// TIA Portal V16 export
// export: Created 2024-12-03T15:41:44.9252202Z, ExportSetting WithReadOnly, DisplayName Totally Integrated Automation Portal, DisplayVersion V16 Update 6, DisplayName TIA Portal Version Control Interface, DisplayVersion V16 Update 2, DisplayName TIA Portal Openness, DisplayVersion V16 Update 6, DisplayName TIA Portal Teamcenter Gateway, DisplayVersion V16, DisplayName SINAMICS Startdrive Advanced, DisplayVersion V16 Update 5, DisplayName SINAMICS Startdrive G130, G150, S120, S150, SINAMICS MV, S210, DisplayVersion V16 Update 5, DisplayName SINAMICS Startdrive G110M, G120, G120C, G120D, G120P, G115D, DisplayVersion V16 Update 5, DisplayName STEP 7 Professional, DisplayVersion V16 Update 6, DisplayName STEP 7 Safety, DisplayVersion V16, DisplayName WinCC Advanced / Unified PC, DisplayVersion V16 Update 6
TYPE "CLXAiPLC_OUT_UDT"
// stored: CreationDate 2021-07-13T07:41:36.2278727Z, InterfaceModifiedDate 2019-12-05T06:54:01.7617053Z, IsConsistent true, LibraryConformanceStatus The object is library-conformant., ModifiedDate 2021-03-27T07:36:50.6363176Z
   STRUCT
      ConveyStopControl { ExternalVisible := 'False'} : Word;   // Writing '1' causes the Stop group to go into STOP state . Writing '2' clears the STOP state
      LeftMDRasDIO : Struct   // Use the MDR as a digital IO
         Reserved0 : Bool;
         Reserved1 : Bool;
         Reserved2 : Bool;
         Reserved3 : Bool;
         Reserved4 : Bool;
         Reserved5 : Bool;
         Reserved6 : Bool;
         SetMotDIO : Bool;   // Write'1' to set the MDR in Digital IO mode
         Reserved8 : Bool;
         DrivePIN4 : Bool;   // Drive the NMOS Transistor of PIN4 on the motor port
         DrivePIN3 : Bool;   // Drive the NMOS Transistor of PIN3 on the motor port
         Reserved11 : Bool;
         Reserved12 : Bool;
         Reserved13 : Bool;
         Reserved14 : Bool;
         Reserved15 : Bool;
      END_STRUCT;
      RightMDRasDIO : Struct   // Use the MDR as a digital IO
         Reserved0 : Bool;
         Reserved1 : Bool;
         Reserved2 : Bool;
         Reserved3 : Bool;
         Reserved4 : Bool;
         Reserved5 : Bool;
         Reserved6 : Bool;
         SetMotDIO : Bool;   // Write'1' to set the MDR in Digital IO mode
         DrivePIN2 : Bool;   // Drive the NMOS Transistor of PIN2 on the motor port
         Reserved9 : Bool;
         DrivePIN3 : Bool;   // Drive the NMOS Transistor of PIN3 on the motor port
         Reserved11 : Bool;
         Reserved12 : Bool;
         Reserved13 : Bool;
         Reserved14 : Bool;
         Reserved15 : Bool;
      END_STRUCT;
      SensorPortsDO { ExternalVisible := 'False'} : Struct   // The Sensor ports PIN2 as digital outputs
         "Reserved[0]" : Bool;
         "Reserved[1]" : Bool;
         "Reserved[2]" : Bool;
         "Reserved[3]" : Bool;
         "Reserved[4]" : Bool;
         "Reserved[5]" : Bool;
         "Reserved[6]" : Bool;
         "Reserved[7]" : Bool;
         DriveLeftPIN2 : Bool;   // Setting this bit drives the Left PIN2 to logical 1
         DriveRightPIN2 : Bool;   // Setting this bit drives the Right PIN2 to logical 1
         "Reserved[10]" : Bool;
         "Reserved[11]" : Bool;
         "Reserved[12]" : Bool;
         SetLeftPIN2asDO : Bool;   // Setting this bit sets the Left PIN2 to be used as Digital Output / 0 = Digital input
         SetRightPIN2asDO : Bool;   // Setting this bit sets the Right PIN2 to be used as Digital Output/ 0 = Digital input
         "Reserved[15]" : Bool;
      END_STRUCT;
      LeftMDRControl { ExternalVisible := 'False'} : Struct   // Run/Stop and Direction control of the Left MDR
         MDR_Direction : Bool;   // 0 = Configured direction /1 = opposite to configured direction
         "Reserved[1]" : Bool;
         "Reserved[2]" : Bool;
         "Reserved[3]" : Bool;
         "Reserved[4]" : Bool;
         "Reserved[5]" : Bool;
         "Reserved[6]" : Bool;
         "Reserved[7]" : Bool;
         Run_MDR : Bool;   // MDR Run = 1 / MDR Stop = 0
         "Reserved[9]" : Bool;
         "Reserved[10]" : Bool;
         "Reserved[11]" : Bool;
         "Reserved[12]" : Bool;
         "Reserved[13]" : Bool;
         "Reserved[14]" : Bool;
         "Reserved[15]" : Bool;
      END_STRUCT;
      LeftMDRBrakeMode { ExternalVisible := 'False'} : Word;   // The Break mode of the Left MDR . 1 = "Normal" / 2 = "Free" / 3 ="Servo break"
      LeftMDR_ServoMode { ExternalVisible := 'False'} : Word;   // 2 = Closed loop servo mode
      RightMDRControl { ExternalVisible := 'False'} : Struct   // Run/Stop and Direction control of the Right MDR
         MDR_Direction : Bool;   // 0 = Configured direction /1 = opposite to configured direction
         "Reserved[1]" : Bool;
         "Reserved[2]" : Bool;
         "Reserved[3]" : Bool;
         "Reserved[4]" : Bool;
         "Reserved[5]" : Bool;
         "Reserved[6]" : Bool;
         "Reserved[7]" : Bool;
         Run_MDR : Bool;   // MDR Run = 1 / MDR Stop = 0
         "Reserved[9]" : Bool;
         "Reserved[10]" : Bool;
         "Reserved[11]" : Bool;
         "Reserved[12]" : Bool;
         "Reserved[13]" : Bool;
         "Reserved[14]" : Bool;
         "Reserved[15]" : Bool;
      END_STRUCT;
      RightMDRBrakeMode { ExternalVisible := 'False'} : Word;   // The Break mode of the Right MDR . 1 = "Normal" / 2 = "Free" / 3 ="Servo break"
      RightMDR_ServoMode { ExternalVisible := 'False'} : Word;   // 2 = Closed loop servo mode
      LeftMDRSpeed { ExternalVisible := 'False'} : Int;   // The speed of the MDR in m/s*1000 .The allowed values depend on the Speed code of the MDR .
      RightMDRSpeed { ExternalVisible := 'False'} : Int;   // The speed of the MDR in m/s*1000 .The allowed values depend on the Speed code of the MDR .
      LeftMDRAccel { ExternalVisible := 'False'} : Int;   // The Acceleration of the left MDR given in "mm"
      LeftMDRDeccel { ExternalVisible := 'False'} : Int;   // The Deceleration of the left MDR given in "mm"
      RightMDRAccel { ExternalVisible := 'False'} : Int;   // The Acceleration of the right MDR given in "mm"
      RightMDRDeccel { ExternalVisible := 'False'} : Int;   // The Deceleration of the right MDR given in "mm"
      ClearMDRError { ExternalVisible := 'False'} : Word;   // Writing '1' to this field clears the MDR error .There needs to be a transition from 0 to 1 in order to clear the error .
      StatusToDownstream { ExternalVisible := 'False'} : Word;   // The ZPA status of our Downstream zone can be written here . A ConveyLinx module in ZPA mode can read this and "Wake up " to accept product
      StatusToUpstream { ExternalVisible := 'False'} : Word;   // The ZPA status of our Upstream zone can be written here . A ConveyLinx module in ZPA mode can read this know we have received the product
      SensorPolarity { ExternalVisible := 'False'} : Struct   // From here the polarity of our Left/Right PIN2/PIN4 can be set
         "Reserved[0]" : Bool;
         "Reserved[1]" : Bool;
         "Reserved[2]" : Bool;
         "Reserved[3]" : Bool;
         "Reserved[4]" : Bool;
         "Reserved[5]" : Bool;
         "Reserved[6]" : Bool;
         "Reserved[7]" : Bool;
         Left_Pin2 : Bool;   // Normal polarity = 0 / Inverted polarity = 1
         "Reserved[9]" : Bool;
         Right_Pin2 : Bool;   // Normal polarity = 0 / Inverted polarity = 1
         "Reserved[11]" : Bool;
         Left_Pin4 : Bool;   // Normal polarity = 0 / Inverted polarity = 1
         "Reserved[13]" : Bool;
         Right_Pin4 : Bool;   // Normal polarity = 0 / Inverted polarity = 1
      END_STRUCT;
      TrackingToDownstream { ExternalVisible := 'False'} : DWord;   // This field can be used to send Tracking data to a downstream ZPA mode ConveyLinx
      Reserved { ExternalVisible := 'False'} : Word;
      ServoControlDistanceLeft { ExternalVisible := 'False'} : Int;   // New MDR distance to be traveled in 'mm'
      ServoControlCommandLeft { ExternalVisible := 'False'} : Struct   // Left MDR servo command
         reserve_7 : Byte;
         ResetPulseCount : Bool;   // Set pulse count (position) to zero
         RunToSetpoint : Bool;   // Run motor from current pulse count to setpoint
         reserve_1 : Bool;
         reserve_2 : Bool;
         reserve_3 : Bool;
         reserve_4 : Bool;
         reserve_5 : Bool;
         reserve_6 : Bool;
      END_STRUCT;
      ServoControlDistanceRight { ExternalVisible := 'False'} : Int;   // New MDR distance to be traveled in 'mm'
      ServoControlCommandRight { ExternalVisible := 'False'} : Struct   // Right MDR servo command
         reserve_1 : Byte;
         ResetPulseCount : Bool;   // Set pulse count (position) to zero
         RunToSetpoint : Bool;   // Run motor from current pulse count to setpoint
         reserve_2 : Bool;
         reserve_3 : Bool;
         reserve_4 : Bool;
         reserve_5 : Bool;
         reserve_6 : Bool;
         reserve_7 : Bool;
      END_STRUCT;
      Future { ExternalVisible := 'False'} : Array[27..31] of Word;
   END_STRUCT;
END_TYPE
